FUNCTION_BLOCK ABSTRACT AB_baseController IMPLEMENTS I_craneControl
VAR_INPUT
END_VAR
VAR_OUTPUT
END_VAR
VAR
END_VAR

METHOD ABSTRACT control_crane 
VAR_INPUT
	stInputs	: ST_inputs_analog;
END_VAR
VAR_OUTPUT
	fCylValve	: REAL;
END_VAR
END_METHOD

METHOD controller
VAR_INPUT
	stButtonInputs	: ST_in_digital;
	stAnalogInputs	: ST_inputs_analog;
END_VAR
VAR_OUTPUT
	stOutput	: ST_ValvePos;
END_VAR
stOutput.rCylinderValve := control_crane(stInputs := stAnalogInputs);
END_METHOD

END_FUNCTION_BLOCK

(* stored: Version 1.1.0.1
   POU AB_baseController: Id {74286472-d9c5-40de-9f74-6ca3ec3cf270}, SpecialFunc None
   Method control_crane: Id {71d61f37-1095-4cc3-bdfa-ab184bb54947}
   Method controller: Id {081b883c-1a06-4c9b-8878-e4f7c5a0625f} *)
